{attribute 'qualified_only'}
TYPE E_OffOn :
(
	_invalid := 0,
	
	Off := 1,
	On := 2
) UDINT;
END_TYPE

(* stored: Version 1.1.0.1
   DUT E_OffOn: Id {cd891a78-0f9f-4e6a-a627-0b1d6fff3cb0} *)
